Fanuc KAREL source: kt00589.KL

PROGRAM KT00589
%STACKSIZE=65535
%PRIORITY=65535
%NOLOCKGROUP
VAR
S1 : STRING[80]
S2 : STRING[80]
OUT : STRING[80]
BEGIN
S1='A'
S2='B'
S1='A'
S2='B'
-- UNRESOLVED_PC line 12 opcodes [73 73 7D 75] marker_code=56
END KT00589
